FUNCTION_BLOCK FinProduccionTemporizado
VAR_INPUT
END_VAR
VAR_OUTPUT
END_VAR
VAR	
	RutaHorno:(Ninguna, Linea5, Linea4_Inf,Linea4_Sup, Linea3, Linea2);
	Estado_FPT:(SalGreenCut_Temp, EntSecadero_Temp, SalAirless_Temp, EntSup_Temp, EntInf_Temp);
	intRutaHorno:INT;
END_VAR
VAR RETAIN
	
END_VAR

//Al activar el fin de producción temporizado empezará un ciclo con temporizadores el cual irá desde la prensa a la entrada del horno reseteando los contadores de piezas.
RutaHorno:=intRutaHorno;

END_FUNCTION_BLOCK

(* stored: Version 1.1.0.1, ProductVersion 3.1.4024.12
   POU FinProduccionTemporizado: Id {9763ee12-8e50-438b-98e7-87fbb4066f00}, SpecialFunc None *)
